{attribute addProperty BoxType "EL3314-0000-0016"}
{attribute addProperty Id "TC_Inputs_ChannelAT %I*ARRAY[0..24] OF TC_Inputs_Channel_E5019A8F288360WcStateAT %I*WcState_98A4DF7520.250InfoDataAT %I*InfoData_BC63D37F80100"}
{attribute addProperty CRC "3654527282"}
{attribute addProperty SizeInBites "370"}
{attribute addProperty SizeInBytes "46.25"}
TYPE EL3314_D4A79586 :
STRUCT
	{attribute addProperty Name "TC_Inputs_Channel"}
	TC_Inputs_Channel : ARRAY[0..24] OF TC_Inputs_Channel_E5019A8F;
	{attribute addProperty Name "WcState"}
	WcState : WcState_98A4DF75;
	{attribute addProperty Name "InfoData"}
	InfoData : InfoData_BC63D37F;
END_STRUCT
END_TYPE

(* stored: Version 1.2.0.0, ProductVersion 3.1.4024.9
   DUT EL3314_D4A79586: Id {46b17bcd-ffde-475b-8f89-edfc531cd70d} *)
